PROGRAM main
VAR
	PushBtn AT %IX0.0 : bool;
	LEDBlue AT %QX0.0 : bool;
	LEDGreen AT %QX0.1 : bool;
	LEDYellow AT %QX0.2 : bool;
	LEDRed AT %QX0.3 : bool;
	DebounceTime : time := T#50ms;
	ledNo : int;
	BtnDelay : bool;
	TONBtnDelay : TON;
	BtnTrigger : R_TRIG;
	triggerReset : bool;
	CountUpLEDNo : CTU;
	LEDRed_Active : bool := FALSE;
	LEDYellow_Active : bool := FALSE;
	LEDGreen_Active : bool;
	LEDBlue_Active : bool;
	R_TRIG0 : R_TRIG;
	pulseReset : bool;
END_VAR
  VAR  (* added by the conversion: wires and edge detectors of the diagram *)
    _GT12_OUT : BOOL;
    _GT12_ENO : BOOL;
  END_VAR

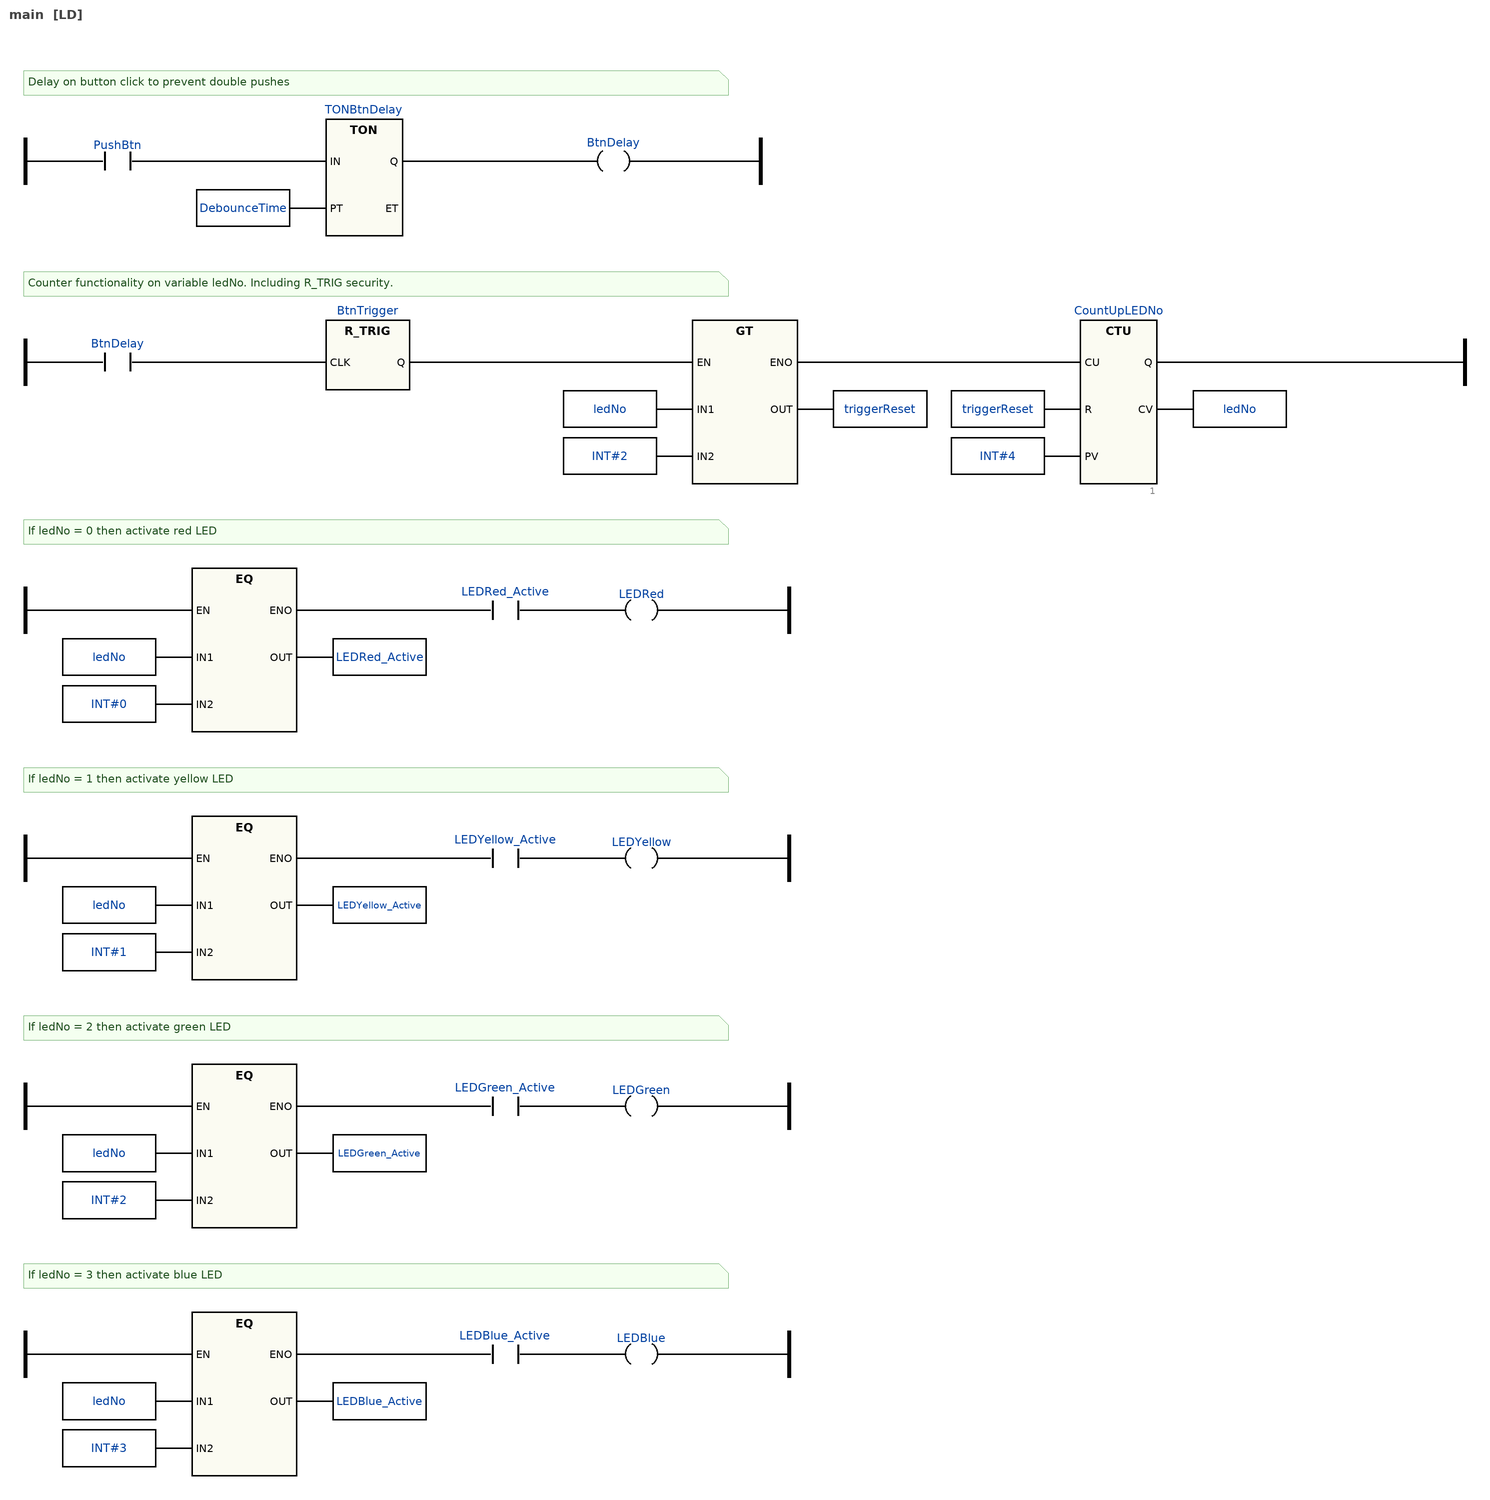
(* LD diagram, written out as Structured Text *)
(* Delay on button click to prevent double pushes *)
(* Counter functionality on variable ledNo. Including R_TRIG security. *)
CountUpLEDNo(CU := _GT12_OUT, R := triggerReset, PV := INT#4);
TONBtnDelay(IN := PushBtn, PT := DebounceTime);
BtnDelay := TONBtnDelay.Q;
BtnTrigger(CLK := BtnDelay);
_GT12_OUT := GT(EN := BtnTrigger.Q, IN1 := ledNo, IN2 := INT#2, ENO => _GT12_ENO);
IF _GT12_ENO THEN triggerReset := _GT12_OUT; END_IF;
ledNo := CountUpLEDNo.CV;
(* If ledNo = 0 then activate red LED *)
LEDRed := LEDRed_Active;
LEDRed_Active := ledNo = INT#0;
(* If ledNo = 1 then activate yellow LED *)
LEDYellow := LEDYellow_Active;
LEDYellow_Active := ledNo = INT#1;
(* If ledNo = 2 then activate green LED *)
LEDGreen := LEDGreen_Active;
LEDGreen_Active := ledNo = INT#2;
(* If ledNo = 3 then activate blue LED *)
LEDBlue := LEDBlue_Active;
LEDBlue_Active := ledNo = INT#3;
END_PROGRAM
